{attribute addProperty BoxType "EJ2918-0000-0017"}
{attribute addProperty Id "FSoE_CommandUSINT811FSOUT_Module_1_Module_FaultBIT10.1251FSOUT_Module_2_Module_FaultBIT10.1251FSoE_CRC_000UINT1623FSoE_Connection_IDUINT1622"}
{attribute addProperty CRC "3786181221"}
{attribute addProperty SizeInBites "48"}
{attribute addProperty SizeInBytes "6"}
TYPE FSOE_E1AC8A65 :
STRUCT
	{attribute addProperty Name "FSoE_Command"}
	FSoE_Command : USINT;
	{attribute addProperty Name "FSOUT_Module_1_Module_Fault"}
	FSOUT_Module_1_Module_Fault : BIT;
	{attribute addProperty Name "FSOUT_Module_2_Module_Fault"}
	FSOUT_Module_2_Module_Fault : BIT;
	{attribute 'hide'}
	reserve_1_BIT_0 : BIT;
	{attribute 'hide'}
	reserve_1_BIT_1 : BIT;
	{attribute 'hide'}
	reserve_1_BIT_2 : BIT;
	{attribute 'hide'}
	reserve_1_BIT_3 : BIT;
	{attribute 'hide'}
	reserve_1_BIT_4 : BIT;
	{attribute 'hide'}
	reserve_1_BIT_5 : BIT;
	{attribute addProperty Name "FSoE_CRC_000"}
	FSoE_CRC_000 : UINT;
	{attribute addProperty Name "FSoE_Connection_ID"}
	FSoE_Connection_ID : UINT;
END_STRUCT
END_TYPE

(* stored: Version 1.2.0.0, ProductVersion 3.1.4024.9
   DUT FSOE_E1AC8A65: Id {07988a48-e972-4809-89c3-b81de732639c} *)
